FUNCTION_BLOCK CROSSCOMM_SENDER_171EE79FA21950F0E (* Service Interface Function Block Type *)
  (* Standard: 61499-2 *)
  (* Version 0.0, 9/22/2017, bababen, nxtControl GmbH, template *)
  PACKAGE Main;
  (* Compiler Cpp nxtControl builtin 1.0 *)
  {SET_ATTRIBUTE(Runtime.FBType.ImplementingType, Runtime.System#DYNGEN_CROSSCOMM_SENDER)}
  {SET_ATTRIBUTE(Configuration.GenericFBType.InterfaceParams, Runtime.System#<InterfaceList> <EventInputs> <Event Name="LIFT_RETRACT" /> <Event Name="LIFT_EXTEND" /> </EventInputs> <InputVars /> </InterfaceList>)}
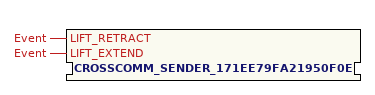
  EVENT_INPUT
    LIFT_RETRACT;
    LIFT_EXTEND;
  END_EVENT
  EC_STATES
    START;
  END_STATES
END_FUNCTION_BLOCK
